(* PLC project Mock Project For Development, Desconhecido Mock Product 1 *)
(* stored: creationDateTime 2023-10-30T11:57:23, modificationDateTime 2023-10-30T12:02:14 *)

(* Program0 mock for development *)
PROGRAM program0
  VAR
    LocalVar0 : DINT := 0;
  END_VAR

            Lorem ipsum dolor sit amet, consectetur adipiscing elit.
Ut interdum sit amet purus id accumsan. Morbi dictum vel nulla et accumsan.
Fusce egestas convallis neque ut elementum. Sed placerat nunc vitae sem pretium dapibus.
Nullam auctor luctus turpis, et consectetur velit accumsan nec. Nullam ut convallis libero,
sed vehicula elit. Suspendisse pretium diam quis massa venenatis, sed dictum purus tincidunt.
Aliquam blandit auctor eros at ornare. Aliquam a mollis neque, placerat convallis lorem.
Proin nec fringilla lectus, vel tincidunt justo. Morbi pretium metus a auctor porta.
Suspendisse imperdiet nulla in nibh blandit, id convallis nulla ullamcorper.
In placerat augue odio, tempor ultrices leo fringilla a.
Praesent purus eros, tempor vitae dolor eget, fringilla tincidunt enim.
          
END_PROGRAM

(* Function0 mock for development *)
FUNCTION function0 : BOOL
  VAR
    LocalVar1 : DINT := 1;
  END_VAR

            Lorem ipsum dolor sit amet, consectetur adipiscing elit.
Ut interdum sit amet purus id accumsan. Morbi dictum vel nulla et accumsan.
Fusce egestas convallis neque ut elementum. Sed placerat nunc vitae sem pretium dapibus.
Nullam auctor luctus turpis, et consectetur velit accumsan nec. Nullam ut convallis libero,
sed vehicula elit. Suspendisse pretium diam quis massa venenatis, sed dictum purus tincidunt.
Aliquam blandit auctor eros at ornare. Aliquam a mollis neque, placerat convallis lorem.
Proin nec fringilla lectus, vel tincidunt justo. Morbi pretium metus a auctor porta.
Suspendisse imperdiet nulla in nibh blandit, id convallis nulla ullamcorper.
In placerat augue odio, tempor ultrices leo fringilla a.
Praesent purus eros, tempor vitae dolor eget, fringilla tincidunt enim.
          
END_FUNCTION

CONFIGURATION Config0
  RESOURCE Res0 ON PLC
    TASK task0(INTERVAL := T#20ms, PRIORITY := 0);
    PROGRAM instance0 WITH task0 : program0;
  END_RESOURCE
END_CONFIGURATION
